// TIA Portal project "PLC_Box_Cerebotani" (V19)

(* hardware
DEVICE "S7-1200 station_1"  S7-1200 Station
   slot 0: "Telaio di montaggio_0"  S7-1200 Rack  Rack  V1.0
   slot 1: "PLC_1"  CPU 1215C DC/DC/DC  6ES7 215-1AG40-0XB0  V4.5
DEVICE "HMI_1"  KTP700 Basic PN SIPLUS
   slot 0: "HMI_1"  KTP700 Basic PN SIPLUS  6AG1 123-2GB03-2AX0  17.0.0.0
   slot 1: "HMI_RT_1"  KTP700 Basic PN SIPLUS  6AG1 123-2GB03-2AX0  17.0.0.0
   slot 5: "HMI_1.IE_CP_1"  PROFINET Interface  17.0.0.0
      slot 1: "Interfaccia_1 PROFINET"  PROFINET Interface
         slot 1: "Porta_1"  Port
*)

// ===== PLC "PLC_1"  CPU 1215C DC/DC/DC =====

VAR_GLOBAL   // PLC tag table "IO"
   "DI_00" AT %I0.0 : Bool;
   "DI_01" AT %I0.1 : Bool;
   "DI_02" AT %I0.2 : Bool;
   "DI_03" AT %I0.3 : Bool;
   "DI_04" AT %I0.4 : Bool;
   "DI_05" AT %I0.5 : Bool;
   "DI_06" AT %I0.6 : Bool;
   "DI_07" AT %I0.7 : Bool;
   "DI_08" AT %I1.0 : Bool;
   "DI_09" AT %I1.1 : Bool;
   "DI_10" AT %I1.2 : Bool;
   "DI_11" AT %I1.3 : Bool;
   "DI_12" AT %I1.4 : Bool;
   "DI_13" AT %I1.5 : Bool;
   "DI_14" AT %I1.6 : Bool;
   "DI_15" AT %I1.7 : Bool;
   "DO_00" AT %Q0.0 : Bool;
   "DO_01" AT %Q0.1 : Bool;
   "DO_02" AT %Q0.2 : Bool;
   "DO_03" AT %Q0.3 : Bool;
   "DO_04" AT %Q0.4 : Bool;
   "DO_05" AT %Q0.5 : Bool;
   "DO_06" AT %Q0.6 : Bool;
   "DO_07" AT %Q0.7 : Bool;
   "DO_08" AT %Q1.0 : Bool;
   "DO_09" AT %Q1.1 : Bool;
   "DO_10" AT %Q1.2 : Bool;
   "DO_11" AT %Q1.3 : Bool;
   "DO_12" AT %Q1.4 : Bool;
   "DO_13" AT %Q1.5 : Bool;
   "DO_14" AT %Q1.6 : Bool;
   "DO_15" AT %Q1.7 : Bool;
END_VAR

DATA_BLOCK "DataOra"   // DB2
{ S7_Optimized_Access := 'TRUE' }
VERSION : 0.1
   VAR
      DateTime : DTL;
   END_VAR
BEGIN
END_DATA_BLOCK

DATA_BLOCK "GestioneSWParalelli"   // DB3
{ S7_Optimized_Access := 'TRUE' }
VERSION : 0.1
   VAR
      NumeroPaginaSW : DInt := 1;
   END_VAR
BEGIN
END_DATA_BLOCK

// folder: System blocks/Program resources

DATA_BLOCK "IEC_Timer_0_DB"   // DB1
{ S7_Optimized_Access := 'TRUE' }
AUTHOR : Simatic
FAMILY : IEC
NAME : IEC_TMR
VERSION : 1.0
// stored: InstanceOfName IEC_TIMER
"IEC_TIMER"
BEGIN
END_DATA_BLOCK

// folder: (top level)

FUNCTION "Test_DO" : Void   // FC1, LAD
{ S7_Optimized_Access := 'TRUE' }
VERSION : 0.1
BEGIN

REGION Network 1
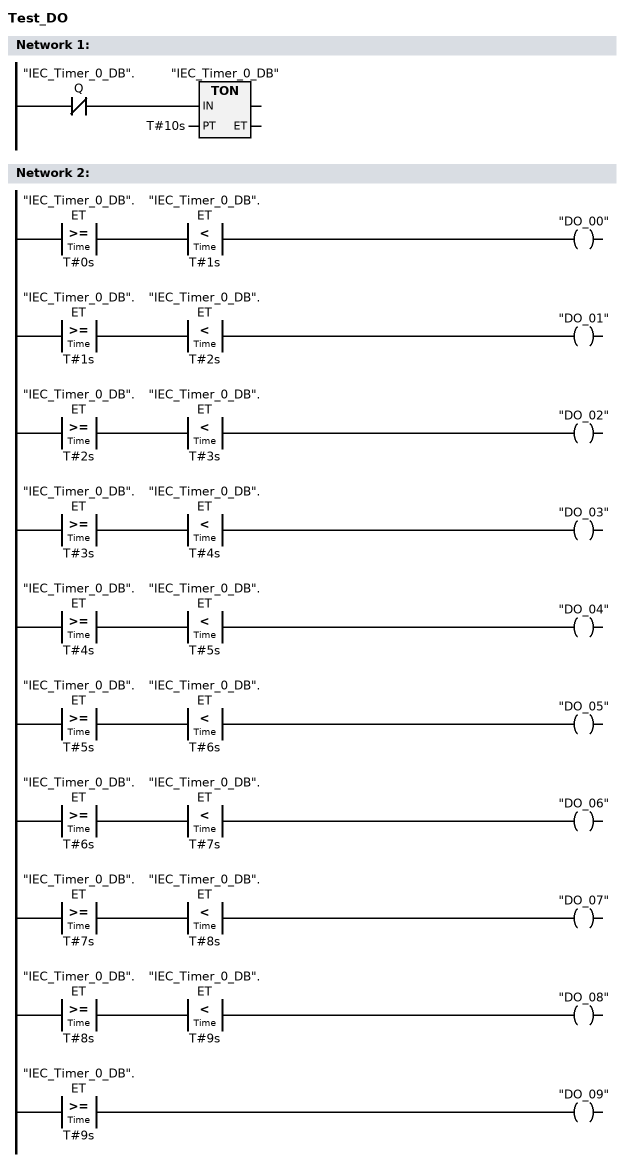
   "IEC_Timer_0_DB".TON(IN := NOT "IEC_Timer_0_DB".Q, PT := T#10s);
END_REGION

REGION Network 2
   RUNG wire#powerrail
      { S7_Templates := "SrcType := Time" } GE_Contact(in1 := "IEC_Timer_0_DB".ET, in2 := T#0s)
      { S7_Templates := "SrcType := Time" } LT_Contact(in1 := "IEC_Timer_0_DB".ET, in2 := T#1s)
      Coil( "DO_00" )
   END_RUNG
   RUNG wire#powerrail
      { S7_Templates := "SrcType := Time" } GE_Contact(in1 := "IEC_Timer_0_DB".ET, in2 := T#1s)
      { S7_Templates := "SrcType := Time" } LT_Contact(in1 := "IEC_Timer_0_DB".ET, in2 := T#2s)
      Coil( "DO_01" )
   END_RUNG
   RUNG wire#powerrail
      { S7_Templates := "SrcType := Time" } GE_Contact(in1 := "IEC_Timer_0_DB".ET, in2 := T#2s)
      { S7_Templates := "SrcType := Time" } LT_Contact(in1 := "IEC_Timer_0_DB".ET, in2 := T#3s)
      Coil( "DO_02" )
   END_RUNG
   RUNG wire#powerrail
      { S7_Templates := "SrcType := Time" } GE_Contact(in1 := "IEC_Timer_0_DB".ET, in2 := T#3s)
      { S7_Templates := "SrcType := Time" } LT_Contact(in1 := "IEC_Timer_0_DB".ET, in2 := T#4s)
      Coil( "DO_03" )
   END_RUNG
   RUNG wire#powerrail
      { S7_Templates := "SrcType := Time" } GE_Contact(in1 := "IEC_Timer_0_DB".ET, in2 := T#4s)
      { S7_Templates := "SrcType := Time" } LT_Contact(in1 := "IEC_Timer_0_DB".ET, in2 := T#5s)
      Coil( "DO_04" )
   END_RUNG
   RUNG wire#powerrail
      { S7_Templates := "SrcType := Time" } GE_Contact(in1 := "IEC_Timer_0_DB".ET, in2 := T#5s)
      { S7_Templates := "SrcType := Time" } LT_Contact(in1 := "IEC_Timer_0_DB".ET, in2 := T#6s)
      Coil( "DO_05" )
   END_RUNG
   RUNG wire#powerrail
      { S7_Templates := "SrcType := Time" } GE_Contact(in1 := "IEC_Timer_0_DB".ET, in2 := T#6s)
      { S7_Templates := "SrcType := Time" } LT_Contact(in1 := "IEC_Timer_0_DB".ET, in2 := T#7s)
      Coil( "DO_06" )
   END_RUNG
   RUNG wire#powerrail
      { S7_Templates := "SrcType := Time" } GE_Contact(in1 := "IEC_Timer_0_DB".ET, in2 := T#7s)
      { S7_Templates := "SrcType := Time" } LT_Contact(in1 := "IEC_Timer_0_DB".ET, in2 := T#8s)
      Coil( "DO_07" )
   END_RUNG
   RUNG wire#powerrail
      { S7_Templates := "SrcType := Time" } GE_Contact(in1 := "IEC_Timer_0_DB".ET, in2 := T#8s)
      { S7_Templates := "SrcType := Time" } LT_Contact(in1 := "IEC_Timer_0_DB".ET, in2 := T#9s)
      Coil( "DO_08" )
   END_RUNG
   RUNG wire#powerrail
      { S7_Templates := "SrcType := Time" } GE_Contact(in1 := "IEC_Timer_0_DB".ET, in2 := T#9s)
      Coil( "DO_09" )
   END_RUNG
   // the same network as SCL:
   "DO_00" := ("IEC_Timer_0_DB".ET >= T#0s) AND ("IEC_Timer_0_DB".ET < T#1s);
   "DO_01" := ("IEC_Timer_0_DB".ET >= T#1s) AND ("IEC_Timer_0_DB".ET < T#2s);
   "DO_02" := ("IEC_Timer_0_DB".ET >= T#2s) AND ("IEC_Timer_0_DB".ET < T#3s);
   "DO_03" := ("IEC_Timer_0_DB".ET >= T#3s) AND ("IEC_Timer_0_DB".ET < T#4s);
   "DO_04" := ("IEC_Timer_0_DB".ET >= T#4s) AND ("IEC_Timer_0_DB".ET < T#5s);
   "DO_05" := ("IEC_Timer_0_DB".ET >= T#5s) AND ("IEC_Timer_0_DB".ET < T#6s);
   "DO_06" := ("IEC_Timer_0_DB".ET >= T#6s) AND ("IEC_Timer_0_DB".ET < T#7s);
   "DO_07" := ("IEC_Timer_0_DB".ET >= T#7s) AND ("IEC_Timer_0_DB".ET < T#8s);
   "DO_08" := ("IEC_Timer_0_DB".ET >= T#8s) AND ("IEC_Timer_0_DB".ET < T#9s);
   "DO_09" := "IEC_Timer_0_DB".ET >= T#9s;
END_REGION
END_FUNCTION

FUNCTION "Test" : Void   // FC2, LAD
{ S7_Optimized_Access := 'TRUE' }
VERSION : 0.1
BEGIN

REGION Network 1
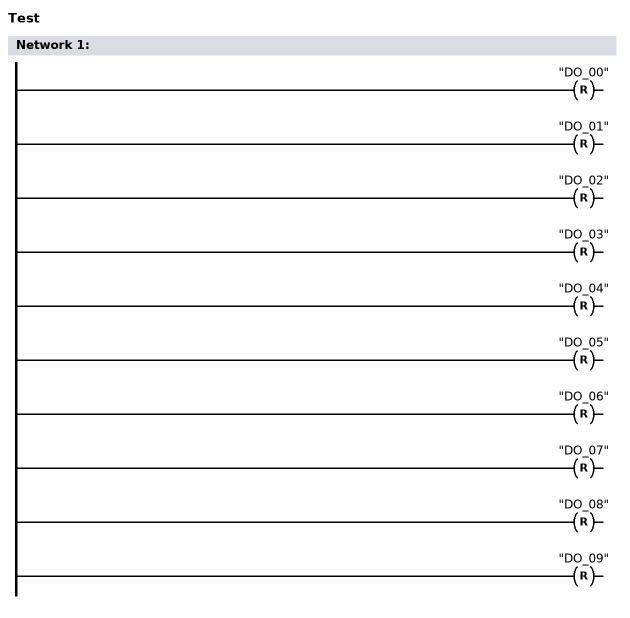
   RUNG wire#powerrail
      R_Coil( "DO_00" )
   END_RUNG
   RUNG wire#powerrail
      R_Coil( "DO_01" )
   END_RUNG
   RUNG wire#powerrail
      R_Coil( "DO_02" )
   END_RUNG
   RUNG wire#powerrail
      R_Coil( "DO_03" )
   END_RUNG
   RUNG wire#powerrail
      R_Coil( "DO_04" )
   END_RUNG
   RUNG wire#powerrail
      R_Coil( "DO_05" )
   END_RUNG
   RUNG wire#powerrail
      R_Coil( "DO_06" )
   END_RUNG
   RUNG wire#powerrail
      R_Coil( "DO_07" )
   END_RUNG
   RUNG wire#powerrail
      R_Coil( "DO_08" )
   END_RUNG
   RUNG wire#powerrail
      R_Coil( "DO_09" )
   END_RUNG
   // the same network as SCL:
   "DO_00" := FALSE;
   "DO_01" := FALSE;
   "DO_02" := FALSE;
   "DO_03" := FALSE;
   "DO_04" := FALSE;
   "DO_05" := FALSE;
   "DO_06" := FALSE;
   "DO_07" := FALSE;
   "DO_08" := FALSE;
   "DO_09" := FALSE;
END_REGION
END_FUNCTION

ORGANIZATION_BLOCK "Main"   // OB1, LAD, ProgramCycle
TITLE = "Main Program Sweep (Cycle)"
{ S7_Optimized_Access := 'TRUE' }
VERSION : 0.1
   VAR_INPUT
      Initial_Call : Bool;   // Initial call of this OB
      Remanence : Bool;   // =True, if remanent data are available
   END_VAR
   VAR_TEMP
      ads : Int;
   END_VAR
BEGIN

REGION Network 1
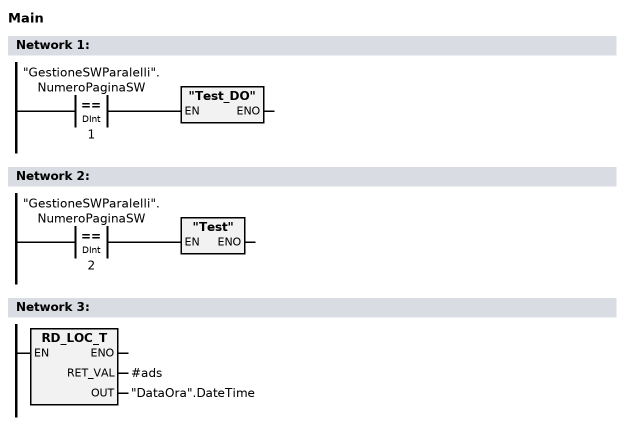
   RUNG wire#powerrail
      { S7_Templates := "SrcType := DInt" } EQ_Contact(in1 := "GestioneSWParalelli".NumeroPaginaSW, in2 := 1)
      "Test_DO"()
   END_RUNG
   // the same network as SCL:
   IF "GestioneSWParalelli".NumeroPaginaSW = 1 THEN "Test_DO"(); END_IF;
END_REGION

REGION Network 2
   RUNG wire#powerrail
      { S7_Templates := "SrcType := DInt" } EQ_Contact(in1 := "GestioneSWParalelli".NumeroPaginaSW, in2 := 2)
      "Test"()
   END_RUNG
   // the same network as SCL:
   IF "GestioneSWParalelli".NumeroPaginaSW = 2 THEN "Test"(); END_IF;
END_REGION

REGION Network 3
   #ads := RD_LOC_T(OUT => "DataOra".DateTime);
END_REGION
END_ORGANIZATION_BLOCK

(* ===== HMI "HMI_RT_1" =====
system functions are stored by id; their names below are inferred from use
connection "HMI_Collegamento_1": ETHERNET, SMART_S7_1200_OMS

HMI tags "Tabella delle variabili standard"
   "Variabile_Numero di pagina" : UInt, internal

HMI tags "IO"
   "DI_00" : Bool = PLC DI_00 AT %I0.0, 100 ms
   "DI_01" : Bool = PLC DI_01 AT %I0.1, 100 ms
   "DI_02" : Bool = PLC DI_02 AT %I0.2, 100 ms
   "DI_03" : Bool = PLC DI_03 AT %I0.3, 100 ms
   "DI_04" : Bool = PLC DI_04 AT %I0.4, 100 ms
   "DI_05" : Bool = PLC DI_05 AT %I0.5, 100 ms
   "DI_06" : Bool = PLC DI_06 AT %I0.6, 100 ms
   "DI_07" : Bool = PLC DI_07 AT %I0.7, 100 ms
   "DI_08" : Bool = PLC DI_08 AT %I1.0, 100 ms
   "DI_09" : Bool = PLC DI_09 AT %I1.1, 100 ms
   "DI_10" : Bool = PLC DI_10 AT %I1.2, 100 ms
   "DI_11" : Bool = PLC DI_11 AT %I1.3, 100 ms
   "DI_12" : Bool = PLC DI_12 AT %I1.4, 100 ms
   "DI_13" : Bool = PLC DI_13 AT %I1.5, 100 ms
   "DI_14" : Bool = PLC DI_14 AT %I1.6, 100 ms
   "DI_15" : Bool = PLC DI_15 AT %I1.7, 100 ms
   "DO_00" : Bool = PLC DO_00 AT %Q0.0, 100 ms
   "DO_01" : Bool = PLC DO_01 AT %Q0.1, 100 ms
   "DO_02" : Bool = PLC DO_02 AT %Q0.2, 100 ms
   "DO_03" : Bool = PLC DO_03 AT %Q0.3, 100 ms
   "DO_04" : Bool = PLC DO_04 AT %Q0.4, 100 ms
   "DO_05" : Bool = PLC DO_05 AT %Q0.5, 100 ms
   "DO_06" : Bool = PLC DO_06 AT %Q0.6, 100 ms
   "DO_07" : Bool = PLC DO_07 AT %Q0.7, 100 ms
   "DO_08" : Bool = PLC DO_08 AT %Q1.0, 100 ms
   "DO_09" : Bool = PLC DO_09 AT %Q1.1, 100 ms
   "DO_10" : Bool = PLC DO_10 AT %Q1.2, 100 ms
   "DO_11" : Bool = PLC DO_11 AT %Q1.3, 100 ms
   "DO_12" : Bool = PLC DO_12 AT %Q1.4, 100 ms
   "DO_13" : Bool = PLC DO_13 AT %Q1.5, 100 ms
   "DO_14" : Bool = PLC DO_14 AT %Q1.6, 100 ms
   "DO_15" : Bool = PLC DO_15 AT %Q1.7, 100 ms

HMI tags "SWParalleli"
   "GestioneSWParalelli_NumeroPaginaSW" : DInt = PLC GestioneSWParalelli.NumeroPaginaSW, 1 s

text list "Elenco testi_Nome della pagina": 1 'Pinout'; 2 'Test'

Template "Modello_1" 800x480
   Button "Esci" at 714,429 size 71x50; TextOff 'Esci'; PictureOff "ExitRuntime_KTP700_Basic_PN_TR"; PictureOn "ExitRuntime_KTP700_Basic_PN_TR"
      on Release: StopRuntime(0)
   Button "Template_Button_1" at 514,429 size 71x50; TextOff 'Text'
   Button "Template_Button_2" at 414,429 size 71x50; TextOff 'Text'
   Button "Template_Button_3" at 314,429 size 71x50; TextOff 'Text'
   Button "Template_Button_4" at 214,429 size 71x50; TextOff 'Text'
   Button "Segnalazioni" at 614,429 size 71x50; TextOff 'Segnalazioni'; PictureOff "AlarmDisplay_KTP700_Basic_PN_TR"; PictureOn "AlarmDisplay_KTP700_Basic_PN_TR"
      on Release: function_ef3f5d25("Finestra delle segnalazioni_Non riconosciuta", -1)
   Button "Pagina iniziale" at 14,429 size 71x50; TextOff 'Pinout'; TextOn 'Pagina iniziale'; PictureOff "NavigateHome_KTP700_Basic_PN_TR"; PictureOn "NavigateHome_KTP700_Basic_PN_TR"
      on Release: ActivateScreen("Pinout", 0)
   SymbolicIOField "Pagina_campo_IO_simbolico" at 93,9 size 600x33; TextOff '0'; TextOn '1'; TextList "Elenco testi_Nome della pagina"
      ProcessValue <- "Variabile_Numero di pagina"
      on Change: ActivateScreenByNumber("Variabile_Numero di pagina", 0)
   DateTimeField "HmiScreenItemData" at 695,25 size 105x25
   DateTimeField "HmiScreenItemData_1" at 695,0 size 105x25
   GraphicView "Logo" at 0,0 size 91x51; Picture "Logo di HMI_1"
   Button "Template_Button_5" at 114,429 size 71x50; TextOff 'Test'
      on Release: ActivateScreen("Test", 0)

screen "Test" 800x480, template "Modello_1"
   on GenerateScreen: SetTag("Variabile_Numero di pagina", 2); SetTag("GestioneSWParalelli_NumeroPaginaSW", 2)

screen "Pinout" 800x480, template "Modello_1"
   on GenerateScreen: SetTag("Variabile_Numero di pagina", 1); SetTag("GestioneSWParalelli_NumeroPaginaSW", 1)
   TextField "HmiScreenItemData_26" at 11,192 size 119x23; Text 'Interruttori'
   Group "Group_1" at 16,218 size 105x95
   TextField "HmiScreenItemData_25" at 11,56 size 119x23; Text 'Pulsanti'
   TextField "HmiScreenItemData_27" at 139,56 size 119x23; Text 'Ausiliari'
   TextField "HmiScreenItemData_28" at 267,56 size 119x23; Text 'Uscite'
   TextField "HmiScreenItemData_9" at 144,82 size 88x23; Text '%I1.0'
   Circle "Cerchio_9" at 226,82 size 23x23
      Appearance <- "DI_08"
   TextField "HmiScreenItemData_10" at 144,106 size 88x23; Text '%I1.1'
   Circle "Cerchio_10" at 226,106 size 23x23
      Appearance <- "DI_09"
   TextField "HmiScreenItemData_11" at 144,130 size 88x23; Text '%I1.2'
   Circle "Cerchio_11" at 226,130 size 23x23
      Appearance <- "DI_10"
   TextField "HmiScreenItemData_12" at 144,154 size 88x23; Text '%I1.3'
   Circle "Cerchio_12" at 226,154 size 23x23
      Appearance <- "DI_11"
   TextField "HmiScreenItemData_13" at 144,178 size 88x23; Text '%I1.4'
   Circle "Cerchio_13" at 226,178 size 23x23
      Appearance <- "DI_12"
   TextField "HmiScreenItemData_14" at 144,202 size 88x23; Text '%I1.5'
   Circle "Cerchio_14" at 226,202 size 23x23
      Appearance <- "DI_13"
   Circle "Cerchio_1" at 98,82 size 23x23
      Appearance <- "DI_00"
   Circle "Cerchio_2" at 98,106 size 23x23
      Appearance <- "DI_01"
   Circle "Cerchio_3" at 98,130 size 23x23
      Appearance <- "DI_02"
   Circle "Cerchio_4" at 98,154 size 23x23
      Appearance <- "DI_03"
   TextField "HmiScreenItemData_1" at 16,82 size 80x23; Text '%I0.0'
   TextField "HmiScreenItemData_2" at 16,106 size 80x23; Text '%I0.1'
   TextField "HmiScreenItemData_3" at 16,130 size 80x23; Text '%I0.2'
   TextField "HmiScreenItemData_4" at 16,154 size 80x23; Text '%I0.3'
   TextField "HmiScreenItemData_15" at 272,82 size 88x23; Text '%Q0.0'
   Circle "Cerchio_15" at 354,82 size 23x23
      Appearance <- "DO_00"
   TextField "HmiScreenItemData_16" at 272,106 size 88x23; Text '%Q0.1'
   Circle "Cerchio_16" at 354,106 size 23x23
      Appearance <- "DO_01"
   TextField "HmiScreenItemData_17" at 272,130 size 88x23; Text '%Q0.2'
   Circle "Cerchio_17" at 354,130 size 23x23
      Appearance <- "DO_02"
   TextField "HmiScreenItemData_18" at 272,154 size 88x23; Text '%Q0.3'
   Circle "Cerchio_18" at 354,154 size 23x23
      Appearance <- "DO_03"
   TextField "HmiScreenItemData_19" at 272,178 size 88x23; Text '%Q0.4'
   Circle "Cerchio_19" at 354,178 size 23x23
      Appearance <- "DO_04"
   TextField "HmiScreenItemData_20" at 272,202 size 88x23; Text '%Q0.5'
   Circle "Cerchio_20" at 354,202 size 23x23
      Appearance <- "DO_05"
   TextField "HmiScreenItemData_21" at 272,226 size 88x23; Text '%Q0.6'
   Circle "Cerchio_21" at 354,226 size 23x23
      Appearance <- "DO_06"
   TextField "HmiScreenItemData_22" at 272,250 size 88x23; Text '%Q0.7'
   Circle "Cerchio_22" at 354,250 size 23x23
      Appearance <- "DO_07"
   TextField "HmiScreenItemData_23" at 272,274 size 88x23; Text '%Q1.0'
   Circle "Cerchio_23" at 354,274 size 23x23
      Appearance <- "DO_08"
   TextField "HmiScreenItemData_24" at 272,298 size 88x23; Text '%Q1.1'
   Circle "Cerchio_24" at 354,298 size 23x23
      Appearance <- "DO_09"
   TextField "HmiScreenItemData_29" at 457,42 size 303x122; Text 'Modello CPU: 1215C DC/DC/DC 6ES7 215-1AG40-0XB0 V4.5'
   TextField "HmiScreenItemData_30" at 457,139 size 303x122; Text 'Modello HMI: KTP700 Basic PN SIPLUS 6AG1 123-2GB03-2AX0 V17.0'
   TextField "HmiScreenItemData_31" at 422,236 size 374x122; Text 'Programma Base: github.com/Filippo-Gambioli/PLC_Box_Cerebotani'
   GraphicView "Vista grafica_1" at 566,334 size 86x82; Picture "Immagine github gambioli"
   TextField "HmiScreenItemData_5" at 16,218 size 104x23; Text '%I0.4'
   Circle "Cerchio_5" at 98,218 size 23x23
      Appearance <- "DI_04"
   TextField "HmiScreenItemData_6" at 16,242 size 104x23; Text '%I0.5'
   Circle "Cerchio_6" at 98,242 size 23x23
      Appearance <- "DI_05"
   Circle "Cerchio_7" at 98,266 size 23x23
      Appearance <- "DI_06"
   Circle "Cerchio_8" at 98,290 size 23x23
      Appearance <- "DI_07"
   TextField "HmiScreenItemData_8" at 16,290 size 104x23; Text '%I0.7'
   TextField "HmiScreenItemData_7" at 16,266 size 104x23; Text '%I0.6'
*)